(* IEC 61131-3 sources: Elmo_Master/Lasal_PRG/MotionTCPDemo/Class/_SigTCPComReceive, 1 file *)

(* ---- _SigTCPComReceive.st ---- *)
(*!
<Class
	Name               = "_SigTCPComReceive"
	Revision           = "1.1"
	RealtimeTask       = "false"
	CyclicTask         = "false"
	BackgroundTask     = "true"
	Sigmatek           = "true"
	OSInterface        = "false"
	HighPriority       = "false"
	Automatic          = "false"
	UpdateMode         = "Prescan"
	SharedCommandTable = "true"
	Objectsize         = "(600,240)"
	Comment            = "Receiving data via TCP communication class. &#13;&#10;&#13;&#10;This class works in combination with the class _SigTCPDataManager and is used to receive data. &#13;&#10;&#13;&#10;Program changes in this class should be considered to be also done in class TCPComReceive.">
	<Channels>
		<Server Name="ClassSvr" Visualized="false" Initialize="false" WriteProtected="true" Retentive="false" Comment="This server can be used to call the global methods of the class."/>
		<Server Name="RecvCnt" Visualized="false" Initialize="false" WriteProtected="false" Retentive="false" Comment="Counter for received data blocks."/>
		<Server Name="SourceID" Visualized="false" Initialize="true" WriteProtected="true" Retentive="false" Comment="Source ID of the TCP-Communication. &#13;&#10;This ID must be the same as the Server DestinationID &#13;&#10;of the _SigTCPComSend from where the data are sent."/>
		<Client Name="_SigTCPDataManager" Required="true" Internal="false" Comment="Connection to communication data manager."/>
	</Channels>
	<RevDoku>
		<Owner Company="Sigmatek"/>
		<Dokumentation Revision="1.1" Date="2025-10-06" Author="KaiAnd" Company="Sigmatek" Description="-- Optimized comments and style&#13;&#10;-- A background task prototype has been implemented (for use in derivations)."/>
		<Dokumentation Revision="1.0" Date="2025-09-24" Author="SchMar2" Company="Sigmatek" Description="New class started from class TCPComReceive V1.0"/>
	</RevDoku>
</Class>
*)
_SigTCPComReceive : CLASS
  //Servers:
	ClassSvr 	: SvrChCmd_DINT;
	SourceID 	: SvrCh_DINT;
	RecvCnt 	: SvrCh_DINT;
  //Clients:
	_SigTCPDataManager 	: CltChCmd__SigTCPDataManager;
  //Variables:
  //Functions:
				//! <Function Comment="Initializations" Name="Init"/>
	FUNCTION VIRTUAL GLOBAL Init;
				//! <Function Comment="Background Task" Name="Background"/>
	FUNCTION VIRTUAL GLOBAL Background
		VAR_INPUT
			EAX 	: UDINT;
		END_VAR
		VAR_OUTPUT
			state (EAX) 	: UDINT;
		END_VAR;
				//! <Function Comment="Is called whenever data is received. &#13;&#10;Overwrite this method to process data. &#13;&#10;NOTE: If the optional CMD parameter is used when sending, the method CallBackReciverCMD() has to be used for receiving in order to correctly receive the CMD parameter." Name="CallBackReceiver"/>
	FUNCTION VIRTUAL GLOBAL CallBackReceiver
		VAR_INPUT
			DestinationID 	: DINT;			//! <Variable Comment="ID of Destination.&#13;&#10;ID like in the send object of the remote station in DestinationID." Name="CallBackReceiver.DestinationID"/>
			SourceID 	: DINT;			//! <Variable Comment="ID of Source.&#13;&#10;ID like in the send object of the remote station in SourceID." Name="CallBackReceiver.SourceID"/>
			size 	: UDINT;			//! <Variable Comment="Length of the data received in bytes" Name="CallBackReceiver.size"/>
			pdata 	: ^USINT;			//! <Variable Comment="Pointer to received data" Name="CallBackReceiver.pdata"/>
		END_VAR
		VAR_OUTPUT
			retcode 	: BOOL;			//! <Variable Comment="TRUE = successfully received = _MNG_Recived &#13;&#10;FALSE = Error in receiving = _MNG_GlobalReciveError&#13;&#10;&#13;&#10;Here you can influence how to react on received data packets. &#13;&#10;If FALSE is returned here, an error is triggered in the sending station (see CallbackJobState in the documentation of the class _SigTCPComSend). " Name="CallBackReceiver.retcode"/>
		END_VAR;
				//! <Function Comment="Overwrite this method in order to receive messages including the optional CMD parameter." Name="CallBackReciverCMD"/>
	FUNCTION VIRTUAL GLOBAL CallBackReciverCMD
		VAR_INPUT
			DestinationID 	: DINT;			//! <Variable Comment="ID of Destination.&#13;&#10;ID like in the send object of the remote station in DestinationID." Name="CallBackReciverCMD.DestinationID"/>
			SourceID 	: DINT;			//! <Variable Comment="ID of Source.&#13;&#10;ID like in the send object of the remote station in SourceID." Name="CallBackReciverCMD.SourceID"/>
			size 	: UDINT;			//! <Variable Comment="Length of the data received in bytes" Name="CallBackReciverCMD.size"/>
			pdata 	: ^USINT;			//! <Variable Comment="Pointer to received data" Name="CallBackReciverCMD.pdata"/>
			OptCMD 	: USINT;			//! <Variable Comment="Optional CMD parameter" Name="CallBackReciverCMD.OptCMD"/>
		END_VAR
		VAR_OUTPUT
			retcode 	: BOOL;			//! <Variable Comment="TRUE = successfully received = _MNG_Recived &#13;&#10;FALSE = Error in receiving = _MNG_GlobalReciveError&#13;&#10;&#13;&#10;Here you can influence how to react on received data packets. &#13;&#10;If FALSE is returned here, an error is triggered in the sending station (see CallbackJobState in the documentation of the class _SigTCPComSend). " Name="CallBackReciverCMD.retcode"/>
		END_VAR;
  //Tables:
	FUNCTION @STD
		VAR_OUTPUT
			ret_code	: CONFSTATES;
		END_VAR;
	FUNCTION GLOBAL TAB @CT_;
END_CLASS;

#pragma usingLtd _SigTCPDataManager

//********************************************************************
// Prototype of callbackmethod
//********************************************************************
FUNCTION GLOBAL CallBackReceiverFnc_SigTCPComReceive
	VAR_INPUT
		pthis 	: ^void;
		DestinationID 	: DINT;
		SourceID 	: DINT;
		size 	: UDINT;
		pdata 	: ^USINT;
	END_VAR
  var_output
    retcode : bool;
  end_var

  retcode := pthis$^_SigTCPComReceive^.CallBackReceiver(DestinationID, SourceID, size, pdata);
  pthis$^_SigTCPComReceive^.RecvCnt +=1;

END_FUNCTION

//********************************************************************
// init method
// connect the receiver do datamanager
//********************************************************************
FUNCTION VIRTUAL GLOBAL _SigTCPComReceive::Init

  if (_FirstScan) then

     // Register as a reception class
    if _SigTCPDataManager.ConnectReciver( udID      := SourceID,
                                          pThis     := this,
                                          pCallback := #CallBackReceiverFnc_SigTCPComReceive()) <> 1 then

      TRACE("_SigTCPComReceive::Init(): Error at login of receiving class");
      ClassSvr := ERROR;
    end_if;

  end_if;

END_FUNCTION

//********************************************************************
// Background Task Prototype
//********************************************************************
FUNCTION VIRTUAL GLOBAL _SigTCPComReceive::Background
	VAR_INPUT
		EAX 	: UDINT;
	END_VAR
	VAR_OUTPUT
		state (EAX) 	: UDINT;
	END_VAR

	state := READY;

END_FUNCTION

//********************************************************************
// callbackmethod of receiver
//********************************************************************
FUNCTION VIRTUAL GLOBAL _SigTCPComReceive::CallBackReceiver
	VAR_INPUT
		DestinationID 	: DINT;
		SourceID 	: DINT;
		size 	: UDINT;
		pdata 	: ^USINT;
	END_VAR
	VAR_OUTPUT
		retcode 	: BOOL;
	END_VAR

  retcode := CallBackReciverCMD(DestinationID:=(DestinationID AND 16#00FFFFFF),
                                SourceID:=SourceID,
                                size:=size,
                                pdata:=pdata,
                                OptCMD:= to_usint((DestinationID$udint AND 16#FF000000) shr 24)  );

END_FUNCTION

//********************************************************************
// callbackmethod to handle the data
//********************************************************************
FUNCTION VIRTUAL GLOBAL _SigTCPComReceive::CallBackReciverCMD
	#pragma warning(disable: 73);
  VAR_INPUT
		DestinationID 	: DINT;
		SourceID 	: DINT;
		size 	: UDINT;
		pdata 	: ^USINT;
		OptCMD 	: USINT;
	END_VAR
	VAR_OUTPUT
		retcode 	: BOOL;
	END_VAR
  #pragma warning(default: 73);

  // received data
  retcode := TRUE;

END_FUNCTION
